TYPE ST_MC_Reset:
STRUCT
	
	CMD_Execute	: 	BOOL;
	
	Done		: 	BOOL;
	Busy		:	BOOL;
	Error		:	BOOL;
	ErrrorID	:	UDINT;	

END_STRUCT
END_TYPE

(* stored: Version 1.1.0.1, ProductVersion 3.1.4024.11
   DUT ST_MC_Reset: Id {7fd3f433-9366-4c61-8edb-479e3cfc45aa} *)
